// TIA Portal V16 export
// export: Created 2023-09-11T12:14:55.1179028Z, ExportSetting WithDefaults, DisplayName Totally Integrated Automation Portal, DisplayVersion V16 Update 6, DisplayName TIA Portal Version Control Interface, DisplayVersion V16 Update 2, DisplayName TIA Portal Openness, DisplayVersion V16 Update 6, DisplayName STEP 7 Professional, DisplayVersion V16 Update 6, DisplayName STEP 7 Safety, DisplayVersion V16, DisplayName WinCC Advanced, DisplayVersion V16 Update 6
FUNCTION "06_M_Switch of signal source of pressure" : Void   // FC5, LAD
{ S7_Optimized_Access := 'TRUE' }
AUTHOR : rtecmer
VERSION : 0.1
// Przęłączanie sygnału źródła ciśnienia zależnie od wybranej strategi: 
// 0- wyłączone, 1- Dosilanie, 2- Przetłączanie, 3- Automat, 4- Ręczne
// stored: AutoNumber true, IsIECCheckEnabled false, SetENOAutomatically false, UDAEnableTagReadback false
   VAR_TEMP   // added for the SCL form of the ladder/FBD networks
      _w1 : Bool;
   END_VAR
BEGIN

REGION Network 1: Filtr Kolmana
   // "switch_kolman" - jeśli 1 to wyłączony jeśli 0 - załączony
END_REGION

REGION Network 2: PV do regulatora PI
   // Podajemy sygnał do PI PV
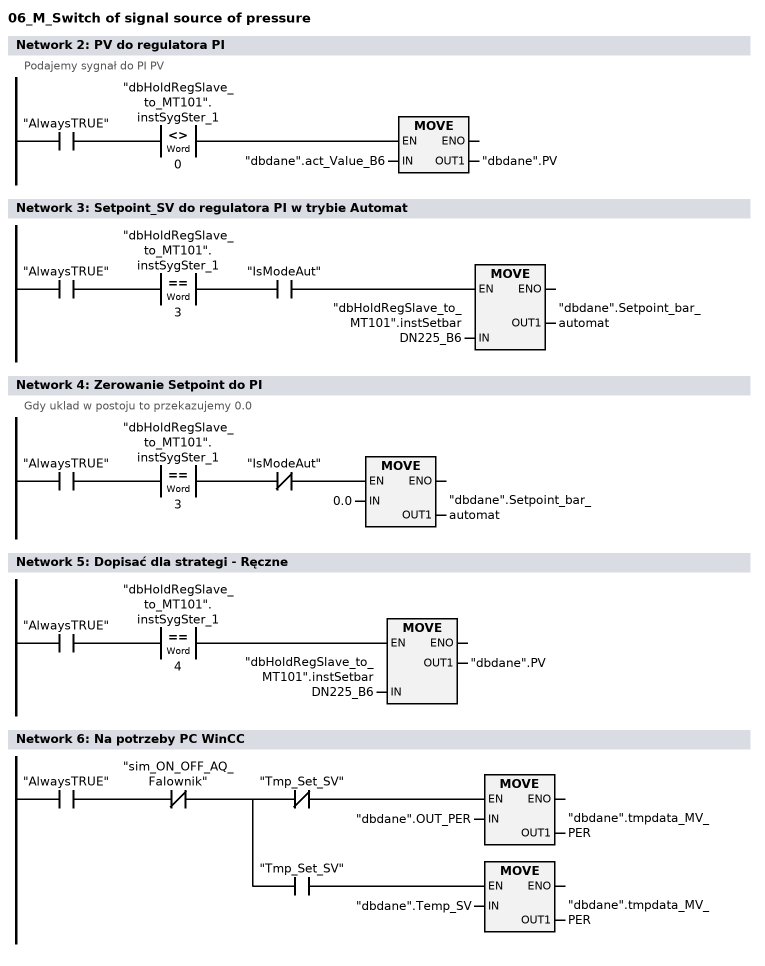
   RUNG wire#powerrail
      Contact( "AlwaysTRUE" )
      { S7_Templates := "SrcType := Word" } NE_Contact(in1 := "dbHoldRegSlave_to_MT101".instSygSter_1, in2 := 0)
      Move(in := "dbdane".act_Value_B6, out1 => "dbdane".PV)
   END_RUNG
   // the same network as SCL:
   IF "AlwaysTRUE" AND ("dbHoldRegSlave_to_MT101".instSygSter_1 <> 0) THEN
       "dbdane".PV := "dbdane".act_Value_B6;
   END_IF;
END_REGION

REGION Network 3: Setpoint_SV do regulatora PI w trybie Automat
   RUNG wire#powerrail
      Contact( "AlwaysTRUE" )
      { S7_Templates := "SrcType := Word" } EQ_Contact(in1 := "dbHoldRegSlave_to_MT101".instSygSter_1, in2 := 3)
      Contact( "IsModeAut" )
      Move(in := "dbHoldRegSlave_to_MT101".instSetbarDN225_B6, out1 => "dbdane".Setpoint_bar_automat)
   END_RUNG
   // the same network as SCL:
   IF "AlwaysTRUE" AND ("dbHoldRegSlave_to_MT101".instSygSter_1 = 3) AND "IsModeAut" THEN
       "dbdane".Setpoint_bar_automat := "dbHoldRegSlave_to_MT101".instSetbarDN225_B6;
   END_IF;
END_REGION

REGION Network 4: Zerowanie Setpoint do PI
   // Gdy uklad w postoju to przekazujemy 0.0
   RUNG wire#powerrail
      Contact( "AlwaysTRUE" )
      { S7_Templates := "SrcType := Word" } EQ_Contact(in1 := "dbHoldRegSlave_to_MT101".instSygSter_1, in2 := 3)
      I_Contact( "IsModeAut" )
      Move(in := 0.0, out1 => "dbdane".Setpoint_bar_automat)
   END_RUNG
   // the same network as SCL:
   IF "AlwaysTRUE" AND ("dbHoldRegSlave_to_MT101".instSygSter_1 = 3) AND NOT "IsModeAut" THEN
       "dbdane".Setpoint_bar_automat := 0.0;
   END_IF;
END_REGION

REGION Network 5: Dopisać dla strategi - Ręczne
   RUNG wire#powerrail
      Contact( "AlwaysTRUE" )
      { S7_Templates := "SrcType := Word" } EQ_Contact(in1 := "dbHoldRegSlave_to_MT101".instSygSter_1, in2 := 4)
      Move(in := "dbHoldRegSlave_to_MT101".instSetbarDN225_B6, out1 => "dbdane".PV)
   END_RUNG
   // the same network as SCL:
   IF "AlwaysTRUE" AND ("dbHoldRegSlave_to_MT101".instSygSter_1 = 4) THEN
       "dbdane".PV := "dbHoldRegSlave_to_MT101".instSetbarDN225_B6;
   END_IF;
END_REGION

REGION Network 6: Na potrzeby PC WinCC
   RUNG wire#powerrail
      Contact( "AlwaysTRUE" )
      I_Contact( "sim_ON_OFF_AQ_Falownik" )
      wire#w1
      I_Contact( "Tmp_Set_SV" )
      { S7_GenerateENO := "TRUE" } Move(in := "dbdane".OUT_PER, out1 => "dbdane".tmpdata_MV_PER)
   END_RUNG
   RUNG wire#w1
      Contact( "Tmp_Set_SV" )
      { S7_GenerateENO := "TRUE" } Move(in := "dbdane".Temp_SV, out1 => "dbdane".tmpdata_MV_PER)
   END_RUNG
   // the same network as SCL:
   #_w1 := "AlwaysTRUE" AND NOT "sim_ON_OFF_AQ_Falownik";
   IF #_w1 AND NOT "Tmp_Set_SV" THEN "dbdane".tmpdata_MV_PER := "dbdane".OUT_PER; END_IF;
   IF #_w1 AND "Tmp_Set_SV" THEN "dbdane".tmpdata_MV_PER := "dbdane".Temp_SV; END_IF;
END_REGION
END_FUNCTION
